// SIMATIC S7-200 SMART project (STEP 7-Micro/WIN SMART), CPU ST60

SYMBOL_TABLE 系统符号
First_Scan_On    SM0.1    // 仅在第一个扫描周期时接通
END_SYMBOL_TABLE

ORGANIZATION_BLOCK MAIN:OB1
TITLE=程序注释
BEGIN
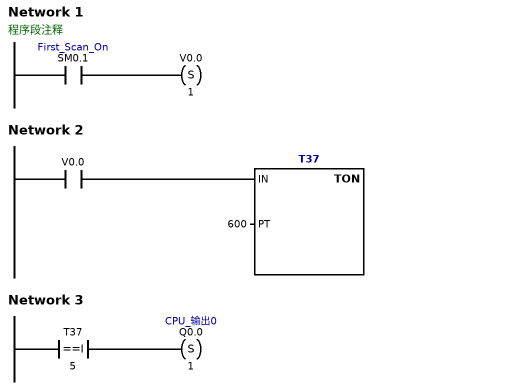
Network 1
// 程序段注释
LD     First_Scan_On:SM0.1
S      V0.0, 1
Network 2
LD     V0.0
TON    T37, 600
Network 3
LDW=   T37, 5
S      CPU_输出0:Q0.0, 1
END_ORGANIZATION_BLOCK
